// SIMATIC STEP 7 (V5.x) project Pneumatic Jacks
// CPU: CPU 314C-2 DP
// station: Hardware
// station: SIMATIC 300(1)
// station: P_ADR_BUS
// program: S7 Program(1)

SYMBOL_TABLE
"start"	I 0.0	BOOL
"Emergency Stop"	I 0.1	BOOL
"Stop all"	M 0.0	BOOL
"Jack1"	Q 0.0	BOOL
"Jack2"	Q 0.1	BOOL
"Jack3"	Q 0.2	BOOL
"Jack4"	Q 0.3	BOOL
END_SYMBOL_TABLE

ORGANIZATION_BLOCK OB 1
TITLE = "Four Pneumatic Jacks"
VERSION : 0.1
VAR_TEMP
  OB1_EV_CLASS : BYTE ;	//Bits 0-3 = 1 (Coming event), Bits 4-7 = 1 (Event class 1)
  OB1_SCAN_1 : BYTE ;	//1 (Cold restart scan 1 of OB 1), 3 (Scan 2-n of OB 1)
  OB1_PRIORITY : BYTE ;	//Priority of OB Execution
  OB1_OB_NUMBR : BYTE ;	//1 (Organization block 1, OB1)
  OB1_RESERVED_1 : BYTE ;	//Reserved for system
  OB1_RESERVED_2 : BYTE ;	//Reserved for system
  OB1_PREV_CYCLE : INT ;	//Cycle time of previous OB1 scan (milliseconds)
  OB1_MIN_CYCLE : INT ;	//Minimum cycle time of OB1 (milliseconds)
  OB1_MAX_CYCLE : INT ;	//Maximum cycle time of OB1 (milliseconds)
  OB1_DATE_TIME : DATE_AND_TIME ;	//Date and time OB1 started
END_VAR
BEGIN
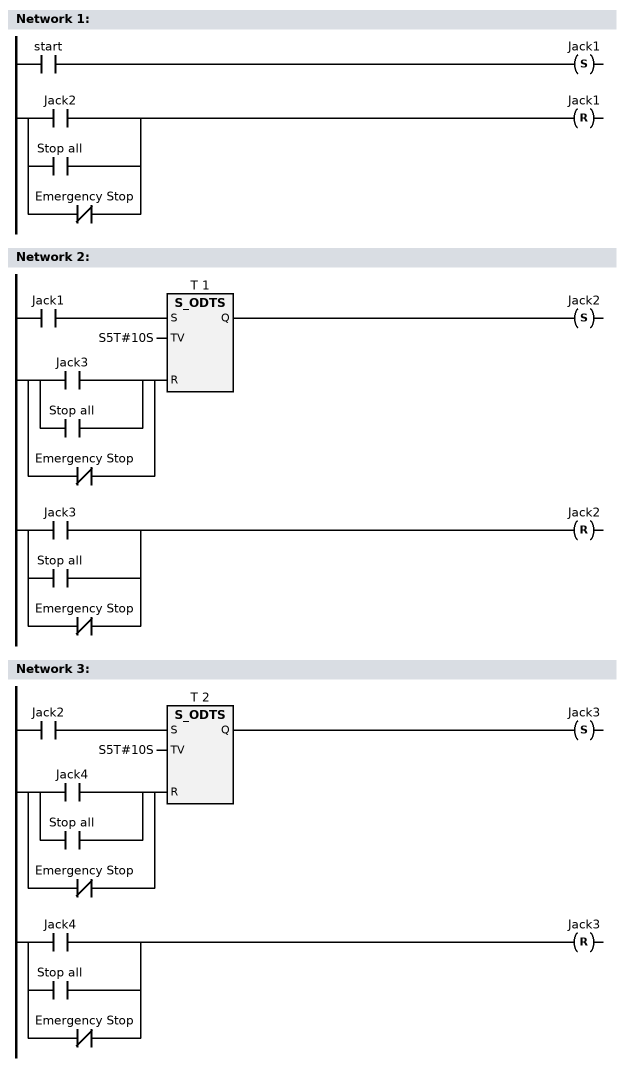
NETWORK
TITLE =
      A     "start";
      S     "Jack1";
      A(;
      O     "Jack2";
      O     "Stop all";
      ON    "Emergency Stop";
      );
      R     "Jack1";
      NOP   0;
NETWORK
TITLE =
      A(;
      A     "Jack1";
      L     S5T#10S;
      SS    T 1;
      A(;
      O     "Jack3";
      O     "Stop all";
      ON    "Emergency Stop";
      );
      R     T 1;
      NOP   0;
      NOP   0;
      A     T 1;
      );
      S     "Jack2";
      A(;
      O     "Jack3";
      O     "Stop all";
      ON    "Emergency Stop";
      );
      R     "Jack2";
      NOP   0;
NETWORK
TITLE =
      A(;
      A     "Jack2";
      L     S5T#10S;
      SS    T 2;
      A(;
      O     "Jack4";
      O     "Stop all";
      ON    "Emergency Stop";
      );
      R     T 2;
      NOP   0;
      NOP   0;
      A     T 2;
      );
      S     "Jack3";
      A(;
      O     "Jack4";
      O     "Stop all";
      ON    "Emergency Stop";
      );
      R     "Jack3";
      NOP   0;
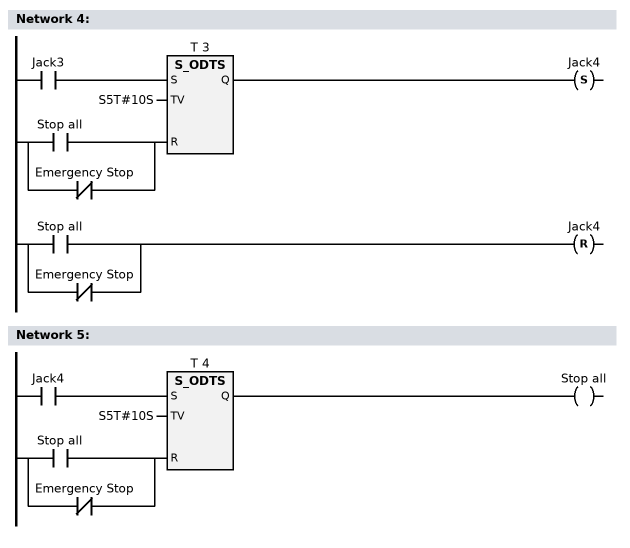
NETWORK
TITLE =
      A(;
      A     "Jack3";
      L     S5T#10S;
      SS    T 3;
      A(;
      O     "Stop all";
      ON    "Emergency Stop";
      );
      R     T 3;
      NOP   0;
      NOP   0;
      A     T 3;
      );
      S     "Jack4";
      A(;
      O     "Stop all";
      ON    "Emergency Stop";
      );
      R     "Jack4";
      NOP   0;
NETWORK
TITLE =
      A     "Jack4";
      L     S5T#10S;
      SS    T 4;
      A(;
      O     "Stop all";
      ON    "Emergency Stop";
      );
      R     T 4;
      NOP   0;
      NOP   0;
      A     T 4;
      =     "Stop all";
END_ORGANIZATION_BLOCK
